% RSLogix 500 project 0c36db70-969f-11e4-95a9-8b42213f1800.RSS, saved by version 8.10.00.24 %
PROJECT "R4 RES"    % processor: MicroLogix 1500 %

PROGRAM FILES
  LAD 2   10 rungs

DATA FILES
  O0 OUTPUT  4 elements
  I1 INPUT  10 elements
  S2 STATUS  66 elements
  B3 BINARY  1 elements
  T4 TIMER  3 elements
  C5 COUNTER  1 elements
  R6 CONTROL  1 elements
  N7 INTEGER  1 elements
  F8 FLOAT  1 elements
  N10   3 elements
  N11   2 elements

LADDER 2
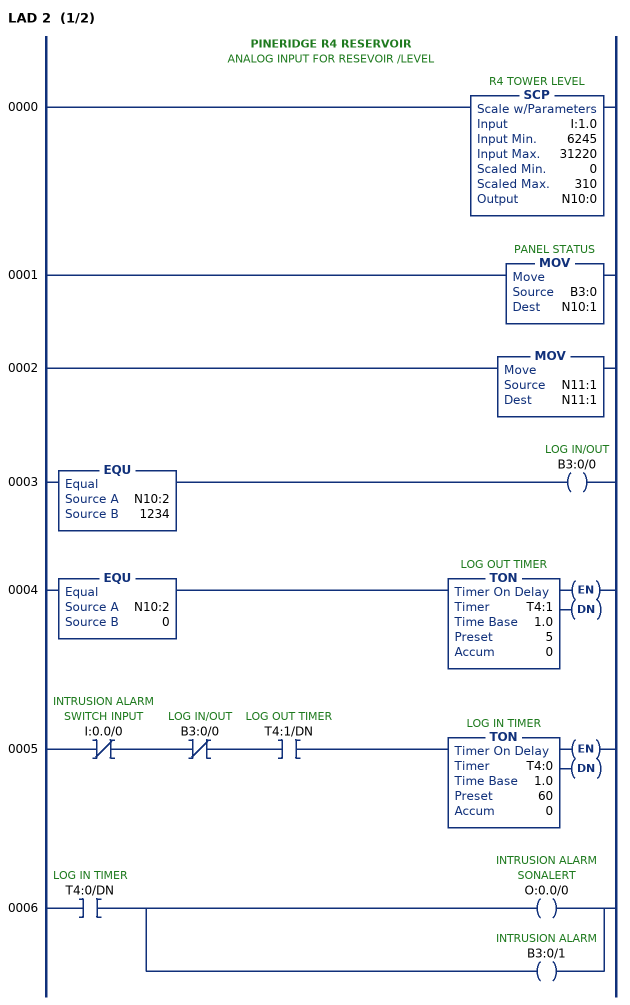
% Rung: 0 %
% TITLE: PINERIDGE R4 RESERVOIR %
% ANALOG INPUT FOR RESEVOIR /LEVEL %
SOR SCP I:1.0 6245 31220 0 310 N10:0 EOR
%   I:1.0  "ANALOG INPUT FOR RESERVOIR LEVEL" %
%   N10:0  "R4 TOWER LEVEL" %
% Rung: 1 %
SOR MOV B3:0 N10:1 EOR
%   B3:0  "INTRUSION ALARM" %
%   N10:1  "PANEL STATUS" %
% Rung: 2 %
SOR MOV N11:1 N11:1 EOR
% Rung: 3 %
SOR EQU N10:2 1234 OTE B3:0/0 EOR
%   B3:0/0  "LOG IN/OUT" %
% Rung: 4 %
SOR EQU N10:2 0 TON T4:1 1.0 5 0 EOR
%   T4:1  "LOG OUT TIMER" %
% Rung: 5 %
SOR XIO I:0.0/0 XIO B3:0/0 XIC T4:1/DN TON T4:0 1.0 60 0 EOR
%   I:0.0/0  "INTRUSION ALARM SWITCH INPUT" %
%   B3:0/0  "LOG IN/OUT" %
%   T4:1  "LOG OUT TIMER" %
%   T4:0  "LOG IN TIMER" %
% Rung: 6 %
SOR XIC T4:0/DN BST OTE O:0.0/0 NXB OTE B3:0/1 BND EOR
%   T4:0  "LOG IN TIMER" %
%   O:0.0/0  "INTRUSION ALARM SONALERT" %
%   B3:0/1  "INTRUSION ALARM" %

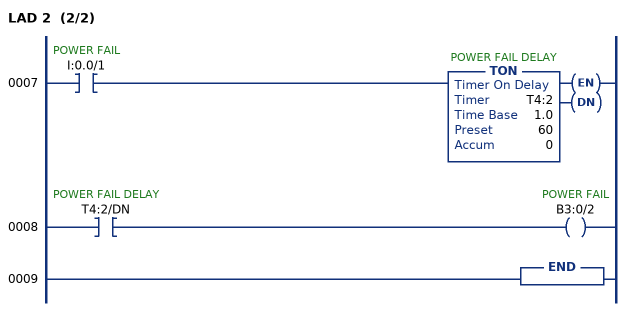
% Rung: 7 %
SOR XIC I:0.0/1 TON T4:2 1.0 60 0 EOR
%   I:0.0/1  "POWER FAIL" %
%   T4:2  "POWER FAIL DELAY" %
% Rung: 8 %
SOR XIC T4:2/DN OTE B3:0/2 EOR
%   T4:2  "POWER FAIL DELAY" %
%   B3:0/2  "POWER FAIL" %
% Rung: 9 %
SOR END EOR

OTHER DOCUMENTED ADDRESSES
  B3:1/0  "INTRUSION ALARM TRIPPED"
  N7:0  "R4 TOWER LEVEL"

DATA TABLE (non-zero values as saved)
DATA B3
% B3:0 % 0X0001
DATA T4
% .PRE .ACC %
% T4:0 % 60 0
% T4:1 % 5 0
% T4:2 % 60 0
DATA N7
% N7:0 % -8
DATA N10
% N10:0 % 253 1 1234
DATA N11
% N11:0 % 5 157
